// TIA Portal project "升降机场景" (V16)

(* hardware
DEVICE "S7-1200 station_1"  S7-1200 Station
   slot 0: "Rack_0"  S7-1200 Rack  Rack  V1.0
   slot 1: "PLC_1"  CPU 1214C DC/DC/DC  6ES7 214-1AG40-0XB0  V4.4
*)

// ===== PLC "PLC_1"  CPU 1214C DC/DC/DC =====

VAR_GLOBAL   // PLC tag table "io表"
   "上料端出口传感器1" AT %I2.0 : Bool;
   "上料端出口传感器2" AT %I2.1 : Bool;
   "上料端出口传感器3" AT %I2.2 : Bool;
   "流水线0末端传感器" AT %I2.3 : Bool;
   "自动模式" AT %I2.4 : Bool;
   "手动模式" AT %I2.5 : Bool;
   "0低" AT %I2.6 : Bool;
   "0高" AT %I2.7 : Bool;
   "1低" AT %I3.0 : Bool;
   "1高" AT %I3.1 : Bool;
   "2低" AT %I3.2 : Bool;
   "2高" AT %I3.3 : Bool;
   "3低" AT %I3.4 : Bool;
   "3高" AT %I3.5 : Bool;
   "启动按钮" AT %I3.6 : Bool;
   "复位按钮" AT %I3.7 : Bool;
   "停止按钮" AT %I4.0 : Bool;
   "急停按钮" AT %I4.1 : Bool;
   "收料端入口传感器" AT %I4.2 : Bool;
   "收料端出口传感器" AT %I4.3 : Bool;
   "FACTORY I/O (Running)" AT %I4.4 : Bool;
   "上料端传送带0" AT %Q2.0 : Bool;
   "上料端传送带1" AT %Q2.1 : Bool;
   "上料端传送带2" AT %Q2.2 : Bool;
   "上料端传送带3" AT %Q2.3 : Bool;
   "出料流水线" AT %Q2.4 : Bool;
   "负载反转" AT %Q2.5 : Bool;
   "负载正转" AT %Q2.6 : Bool;
   "升降机向上" AT %Q2.7 : Bool;
   "升降机向下" AT %Q3.0 : Bool;
   "升降机减速" AT %Q3.1 : Bool;
   "报警器" AT %Q3.2 : Bool;
   "绿色" AT %Q3.3 : Bool;
   "黄色" AT %Q3.4 : Bool;
   "红色" AT %Q3.5 : Bool;
   "蓝色1" AT %Q3.6 : Bool;
   "蓝色2" AT %Q3.7 : Bool;
   "蓝色3" AT %Q4.0 : Bool;
   "绿色1" AT %Q4.1 : Bool;
   "黄色1" AT %Q4.2 : Bool;
   "红色1" AT %Q4.3 : Bool;
   "绿色2" AT %Q4.4 : Bool;
   "黄色2" AT %Q4.5 : Bool;
   "红色2" AT %Q4.6 : Bool;
   "绿色3" AT %Q4.7 : Bool;
   "黄色3" AT %Q5.0 : Bool;
   "红色3" AT %Q5.1 : Bool;
   "显示屏" AT %QD30 : DInt;
END_VAR

VAR_GLOBAL   // PLC tag table "中间变量"
   "启动标志位" AT %M0.0 : Bool;
   "中间变量1" AT %M5.1 : Bool;
   "中间变量2" AT %M5.2 : Bool;
   "中间变量3" AT %M5.3 : Bool;
   "中间变量4" AT %M5.4 : Bool;
   "中间变量5" AT %M5.5 : Bool;
   "中间变量6" AT %M5.6 : Bool;
   "中间变量7" AT %M5.7 : Bool;
   "中间变量8" AT %M6.0 : Bool;
   "中间变量9" AT %M6.1 : Bool;
   "中间变量10" AT %M6.2 : Bool;
   "中间变量11" AT %M6.3 : Bool;
   "中间变量12" AT %M6.4 : Bool;
   "中间变量13" AT %M6.5 : Bool;
   "中间变量14" AT %M6.6 : Bool;
   "中间变量15" AT %M6.7 : Bool;
   "启动升降机" AT %M0.1 : Bool;
   "一楼等待" AT %M0.2 : Bool;
   "一楼延时" AT %M0.3 : Bool;
   "二楼等待" AT %M0.4 : Bool;
   "二楼延时" AT %M0.5 : Bool;
   "三楼等待" AT %M0.6 : Bool;
   "三楼延时" AT %M0.7 : Bool;
   "准备上升" AT %M1.0 : Bool;
   "停止" AT %M1.1 : Bool;
   "准备下降" AT %M1.2 : Bool;
END_VAR

// folder: System blocks/Program resources

DATA_BLOCK "IEC_Timer_0_DB"   // DB1
{ S7_Optimized_Access := 'TRUE' }
AUTHOR : Simatic
FAMILY : IEC
NAME : IEC_TMR
VERSION : 1.0
// stored: InstanceOfName IEC_TIMER
"IEC_TIMER"
BEGIN
END_DATA_BLOCK

DATA_BLOCK "IEC_Timer_0_DB_1"   // DB2
{ S7_Optimized_Access := 'TRUE' }
AUTHOR : Simatic
FAMILY : IEC
NAME : IEC_TMR
VERSION : 1.0
// stored: InstanceOfName IEC_TIMER
"IEC_TIMER"
BEGIN
END_DATA_BLOCK

DATA_BLOCK "IEC_Timer_0_DB_2"   // DB3
{ S7_Optimized_Access := 'TRUE' }
AUTHOR : Simatic
FAMILY : IEC
NAME : IEC_TMR
VERSION : 1.0
// stored: InstanceOfName IEC_TIMER
"IEC_TIMER"
BEGIN
END_DATA_BLOCK

// folder: (top level)

FUNCTION "MHJ-PLC-Lab-Function-S71200" : Void   // FC9000, SCL
{ S7_Optimized_Access := 'TRUE' }
VERSION : 0.1
   VAR_TEMP
      rdTimeReturn : Int;
      outputTime : DTL;
      SyncVal : Byte;
      forVal : Int;
      forVal_2 : Int;
      Value : Byte;
   END_VAR
   VAR CONSTANT
      CompVal : Byte := 16#34;
      Value_01 : Byte := 16#11;
      Value_01_DW : DWord := 16#A165_D992;
      Value_02_DW : DWord := 16#58BE_4401;
   END_VAR
BEGIN

   #Value:=PEEK(area := 16#82,
        dbNumber := 0,
        byteOffset := 511);
   #Value := #Value + 1;

   POKE(area := 16#82,
        dbNumber := 0,
        byteOffset := 511,
        value := #Value);

   POKE(area:=16#81,
        dbNumber:=0,
        byteOffset:=1016,
        value:=#Value_01_DW);
   POKE(area := 16#81,
        dbNumber := 0,
        byteOffset := 1020,
        value := #Value_02_DW);

   POKE(area := 16#81,
        dbNumber := 0,
        byteOffset := 511,
        value := B#16#00);

   FOR #forVal := 0 TO 120 DO
       FOR #forVal_2:=0 TO 10 DO
           #rdTimeReturn:=RD_SYS_T(#outputTime);
           #rdTimeReturn := WR_SYS_T(#outputTime);
           #rdTimeReturn := RD_SYS_T(#outputTime);
           #rdTimeReturn := WR_SYS_T(#outputTime);
       END_FOR;
       #SyncVal:= PEEK(area := 16#81,
                      dbNumber := 0,
                      byteOffset := 511);
       IF #SyncVal = #CompVal THEN
          GOTO M_1;
       END_IF;
   END_FOR;
   RETURN;

   M_1:
   POKE(area := 16#81,
        dbNumber := 0,
        byteOffset := 511,
        value := B#16#0);
END_FUNCTION

ORGANIZATION_BLOCK "Main"   // OB1, LAD, ProgramCycle
TITLE = "Main Program Sweep (Cycle)"
{ S7_Optimized_Access := 'TRUE' }
VERSION : 0.1
   VAR_INPUT
      Initial_Call : Bool;   // Initial call of this OB
      Remanence : Bool;   // =True, if remanent data are available
   END_VAR
   VAR_TEMP   // added for the SCL form of the ladder/FBD networks
      _w1 : Bool;
      _w2 : Bool;
      _w3 : Bool;
   END_VAR
BEGIN

REGION Network 1
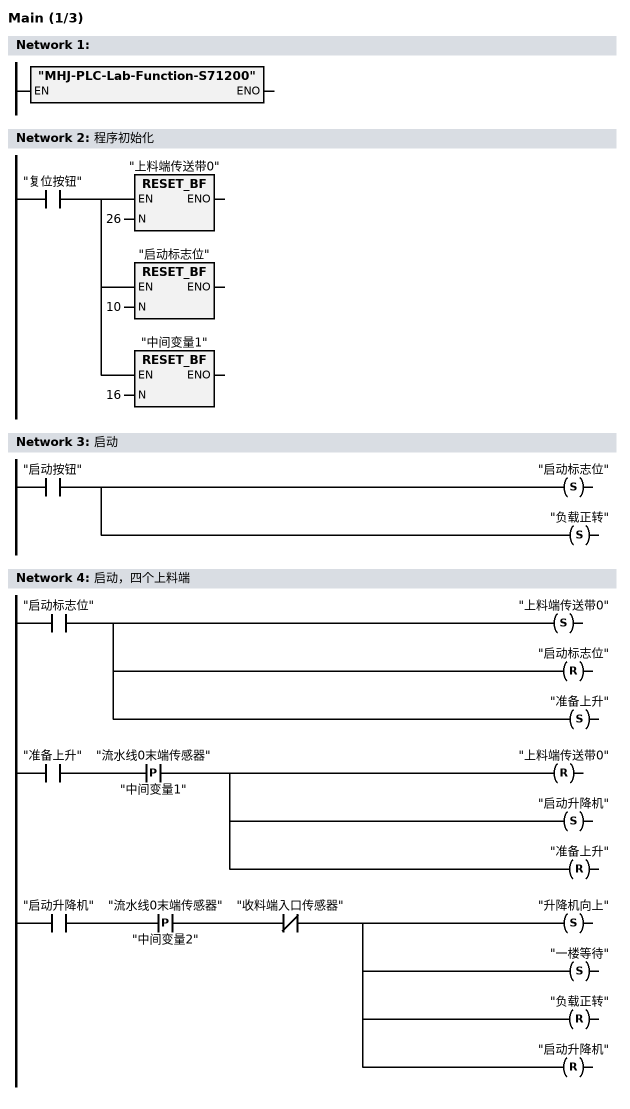
   RUNG wire#powerrail
      "MHJ-PLC-Lab-Function-S71200"()
   END_RUNG
   // the same network as SCL:
   "MHJ-PLC-Lab-Function-S71200"();
END_REGION

REGION Network 2: 程序初始化
   // no SCL statement known for RBitfield: written as a call
   #_w1 := "复位按钮";
   IF #_w1 THEN
       RESET_BF(operand := "上料端传送带0", n := 26);
       RESET_BF(operand := "启动标志位", n := 10);
       RESET_BF(operand := "中间变量1", n := 16);
   END_IF;
END_REGION

REGION Network 3: 启动
   RUNG wire#powerrail
      Contact( "启动按钮" )
      wire#w1
      S_Coil( "启动标志位" )
   END_RUNG
   RUNG wire#w1
      S_Coil( "负载正转" )
   END_RUNG
   // the same network as SCL:
   IF "启动按钮" THEN
       "启动标志位" := TRUE;
       "负载正转" := TRUE;
   END_IF;
END_REGION

REGION Network 4: 启动，四个上料端
   RUNG wire#powerrail
      Contact( "启动标志位" )
      wire#w1
      S_Coil( "上料端传送带0" )
   END_RUNG
   RUNG wire#w1
      R_Coil( "启动标志位" )
   END_RUNG
   RUNG wire#w1
      S_Coil( "准备上升" )
   END_RUNG
   RUNG wire#powerrail
      Contact( "准备上升" )
      P_Contact(operand := "流水线0末端传感器", bit := "中间变量1")
      wire#w2
      R_Coil( "上料端传送带0" )
   END_RUNG
   RUNG wire#w2
      S_Coil( "启动升降机" )
   END_RUNG
   RUNG wire#w2
      R_Coil( "准备上升" )
   END_RUNG
   RUNG wire#powerrail
      Contact( "启动升降机" )
      P_Contact(operand := "流水线0末端传感器", bit := "中间变量2")
      I_Contact( "收料端入口传感器" )
      wire#w3
      S_Coil( "升降机向上" )
   END_RUNG
   RUNG wire#w3
      S_Coil( "一楼等待" )
   END_RUNG
   RUNG wire#w3
      R_Coil( "负载正转" )
   END_RUNG
   RUNG wire#w3
      R_Coil( "启动升降机" )
   END_RUNG
   // the same network as SCL:
   IF "启动标志位" THEN "上料端传送带0" := TRUE; END_IF;
   #_w1 := "启动标志位";
   IF #_w1 THEN
       "启动标志位" := FALSE;
       "准备上升" := TRUE;
   END_IF;
   #_w2 := "准备上升" AND "流水线0末端传感器" AND NOT "中间变量1";   // rising edge of "流水线0末端传感器"
   "中间变量1" := "流水线0末端传感器";
   IF #_w2 THEN
       "上料端传送带0" := FALSE;
       "启动升降机" := TRUE;
       "准备上升" := FALSE;
   END_IF;
   #_w3 := "启动升降机" AND "流水线0末端传感器" AND NOT "中间变量2";   // rising edge of "流水线0末端传感器"
   "中间变量2" := "流水线0末端传感器";
   IF #_w3 AND NOT "收料端入口传感器" THEN
       "升降机向上" := TRUE;
       "一楼等待" := TRUE;
       "负载正转" := FALSE;
       "启动升降机" := FALSE;
   END_IF;
END_REGION

REGION Network 5: 一楼开始
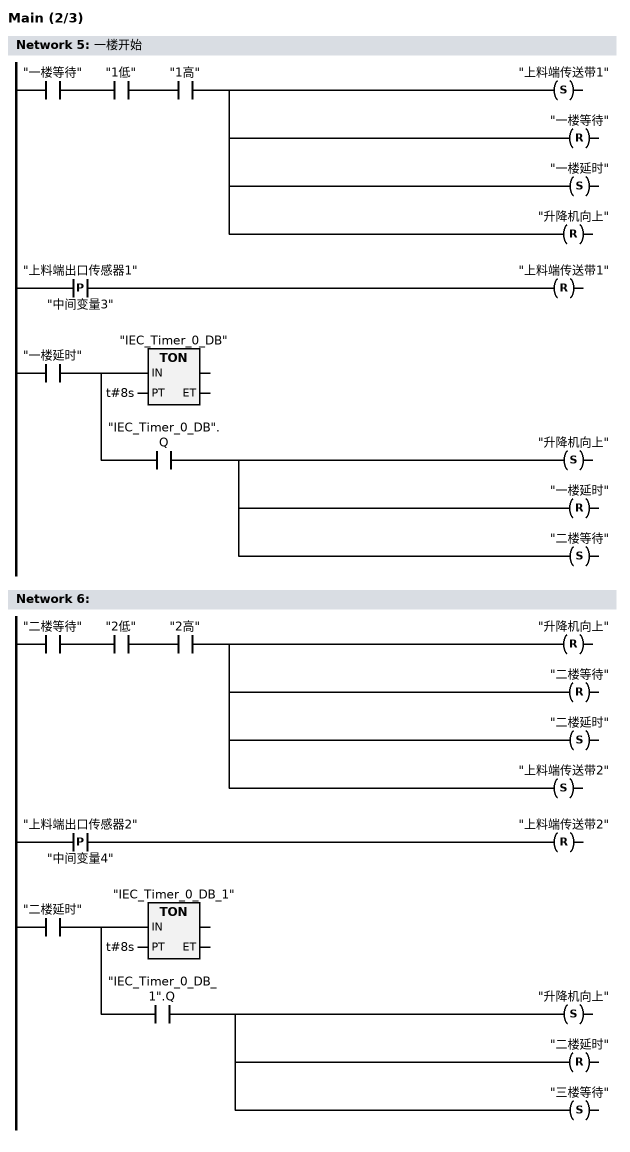
   IF "一楼等待" AND "1低" AND "1高" THEN "上料端传送带1" := TRUE; END_IF;
   #_w1 := "一楼等待" AND "1低" AND "1高";
   IF #_w1 THEN
       "一楼等待" := FALSE;
       "一楼延时" := TRUE;
       "升降机向上" := FALSE;
   END_IF;
   #_w2 := "上料端出口传感器1" AND NOT "中间变量3";   // rising edge of "上料端出口传感器1"
   "中间变量3" := "上料端出口传感器1";
   IF #_w2 THEN "上料端传送带1" := FALSE; END_IF;
   "IEC_Timer_0_DB".TON(IN := "一楼延时", PT := t#8s);
   IF "一楼延时" AND "IEC_Timer_0_DB".Q THEN "升降机向上" := TRUE; END_IF;
   #_w3 := "一楼延时" AND "IEC_Timer_0_DB".Q;
   IF #_w3 THEN
       "一楼延时" := FALSE;
       "二楼等待" := TRUE;
   END_IF;
END_REGION

REGION Network 6
   IF "二楼等待" AND "2低" AND "2高" THEN "升降机向上" := FALSE; END_IF;
   #_w1 := "二楼等待" AND "2低" AND "2高";
   IF #_w1 THEN
       "二楼等待" := FALSE;
       "二楼延时" := TRUE;
       "上料端传送带2" := TRUE;
   END_IF;
   #_w2 := "上料端出口传感器2" AND NOT "中间变量4";   // rising edge of "上料端出口传感器2"
   "中间变量4" := "上料端出口传感器2";
   IF #_w2 THEN "上料端传送带2" := FALSE; END_IF;
   "IEC_Timer_0_DB_1".TON(IN := "二楼延时", PT := t#8s);
   IF "二楼延时" AND "IEC_Timer_0_DB_1".Q THEN "升降机向上" := TRUE; END_IF;
   #_w3 := "二楼延时" AND "IEC_Timer_0_DB_1".Q;
   IF #_w3 THEN
       "二楼延时" := FALSE;
       "三楼等待" := TRUE;
   END_IF;
END_REGION

REGION Network 7
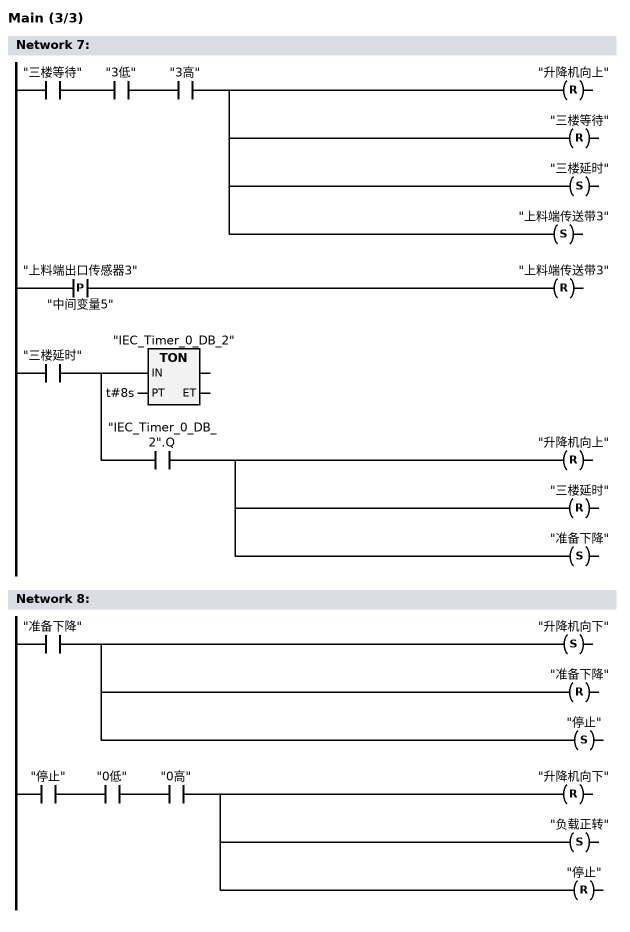
   IF "三楼等待" AND "3低" AND "3高" THEN "升降机向上" := FALSE; END_IF;
   #_w1 := "三楼等待" AND "3低" AND "3高";
   IF #_w1 THEN
       "三楼等待" := FALSE;
       "三楼延时" := TRUE;
       "上料端传送带3" := TRUE;
   END_IF;
   #_w2 := "上料端出口传感器3" AND NOT "中间变量5";   // rising edge of "上料端出口传感器3"
   "中间变量5" := "上料端出口传感器3";
   IF #_w2 THEN "上料端传送带3" := FALSE; END_IF;
   "IEC_Timer_0_DB_2".TON(IN := "三楼延时", PT := t#8s);
   IF "三楼延时" AND "IEC_Timer_0_DB_2".Q THEN "升降机向上" := FALSE; END_IF;
   #_w3 := "三楼延时" AND "IEC_Timer_0_DB_2".Q;
   IF #_w3 THEN
       "三楼延时" := FALSE;
       "准备下降" := TRUE;
   END_IF;
END_REGION

REGION Network 8
   RUNG wire#powerrail
      Contact( "准备下降" )
      wire#w1
      S_Coil( "升降机向下" )
   END_RUNG
   RUNG wire#w1
      R_Coil( "准备下降" )
   END_RUNG
   RUNG wire#w1
      S_Coil( "停止" )
   END_RUNG
   RUNG wire#powerrail
      Contact( "停止" )
      Contact( "0低" )
      Contact( "0高" )
      wire#w2
      R_Coil( "升降机向下" )
   END_RUNG
   RUNG wire#w2
      S_Coil( "负载正转" )
   END_RUNG
   RUNG wire#w2
      R_Coil( "停止" )
   END_RUNG
   // the same network as SCL:
   IF "准备下降" THEN "升降机向下" := TRUE; END_IF;
   #_w1 := "准备下降";
   IF #_w1 THEN
       "准备下降" := FALSE;
       "停止" := TRUE;
   END_IF;
   IF "停止" AND "0低" AND "0高" THEN
       "升降机向下" := FALSE;
       "负载正转" := TRUE;
       "停止" := FALSE;
   END_IF;
END_REGION
END_ORGANIZATION_BLOCK